# EPICS substitutions: ThingyApp/Db/notify.substitutions
file "notify.template"
{
pattern { Sys, 	Dev  		  ,	Attr 		 , Units,	UUID, 	Next}
{ "XF:10IDB",	"{THINGY:001}",	"Temperature", "C",		"201",	"Pressure"}
{ "XF:10IDB",	"{THINGY:001}",	"Pressure",    "hPa",	"202",	"Humidity"}
{ "XF:10IDB",	"{THINGY:001}",	"Humidity",    "%",		"203",	"Button"}

{ "XF:10IDB", 	"{THINGY:001}",	"Button",	   "",		"302",	"Orientation"}

{ "XF:10IDB", 	"{THINGY:001}",	"Orientation", "",		"403",	""}
}
